// TIA Portal V17 export
// export: Created 2024-09-02T12:50:27.4175061Z, ExportSetting WithDefaults, DisplayName Totally Integrated Automation Portal, DisplayVersion V17, DisplayName TIA Portal Openness, DisplayVersion V17, DisplayName TIA Portal Version Control Interface, DisplayVersion V17, DisplayName STEP 7 Professional, DisplayVersion V17, DisplayName STEP 7 Safety, DisplayVersion V17, DisplayName WinCC Professional, DisplayVersion V17
TYPE "TypeSKS_DREH"
// stored: IsFailsafeCompliant false
   STRUCT
      "A" : Struct
         "90Deg" : Bool;
         "0Deg" : Bool;
      END_STRUCT;
      H : Struct
         "90Deg" : Bool;
         "0Deg" : Bool;
      END_STRUCT;
   END_STRUCT;
END_TYPE
